// TIA Portal V18 export
FUNCTION_BLOCK "IR_Heater_Control"   // FB17, LAD
TITLE = Description
{ S7_Optimized_Access := 'TRUE' }
VERSION : 0.1
// How to control and set the IR lamp:
// To turn on the IR lamp the machine needs to be started and the doors closed. Heater setpoint should be set from 0-100 "Heater_Setpoint", lamp should be turned on by "Heater_ON_OFF". The lamp will activate only when the certain conditions are meet (position/direction/time).
// 
// Right now, the signal from NOAH is being send when spreading and the permission for the lamp is being keep in the function block for a certain period of time to enable the lamp on the way back.
// 
// E-STOP - always check!
// 
// Modes:
// 0 - Heating Feedbox/Printbox when spreading and executing the heater on the way back from PLC
// 1 - Heating only on the way back from NOAH
// 
// Safety is based only on timer. Hardware protection should be implemented ASAP (contactor controlled by thermal fuse / thermistor to cut off the power if the temperature exceeds certain level).
// 
// Things to implement:
// - Remote temperature sensor(already purchased some time ago).
// - Heater_MathFunction to operate heater better based on the measured results
// - PID control
// 
// Status:
// Filip 14.12.2022: Added modes to give full control to NOAH (Mode 1) or control heater on the way back from PLC (Mode 0)
// stored: AutoNumber true, IsIECCheckEnabled false, IsRetainMemResEnabled false, MemoryReserve 100, SetENOAutomatically false, UDAEnableTagReadback false
   VAR_INPUT
      MachineNumber : Int;
      Mode : Int := 1;   // 0 - Heating partly from PLC; 1 - Full control from NOAH
      DoorSenor : Bool;
      RollerON { ExternalAccessible := 'False'; ExternalVisible := 'False'; ExternalWritable := 'False'} : Bool;   // General heater safety condition
      Heater_Safety_PDL { ExternalAccessible := 'False'; ExternalVisible := 'False'; ExternalWritable := 'False'} : Real;   // Pulse Duration Limit - set by technician or engineer in charge, don't change
      Heater_PWM_address { ExternalAccessible := 'False'; ExternalVisible := 'False'; ExternalWritable := 'False'} : HW_PWM;   // PLC PWM output address
      Heater_Setpoint { ExternalAccessible := 'False'; ExternalVisible := 'False'; ExternalWritable := 'False'} : Real;
      "E-STOP" { ExternalAccessible := 'False'; ExternalVisible := 'False'; ExternalWritable := 'False'} : Bool;
      Heater_ON_OFF { ExternalAccessible := 'False'; ExternalVisible := 'False'; ExternalWritable := 'False'} : Bool;   // WebDB
      FeedboxHeating : Bool;
      PrintboxHeating : Bool;
      AxisYActualPosition : DInt;
      AxisYActualVelocity : Real;
      FeedboxStartMachine : DInt;
      FeedboxEndMachine : DInt;
      PrintboxStartMachine : DInt;
      PrintboxEndMachine : DInt;
      HeaterTest : Bool;
   END_VAR
   VAR_OUTPUT
      Heater_Output : Bool;
      Heater_Pulse_Duration : Int;
      Heater_Error : Int;
      Heater_Output_Check : Int;
      RollerONWayBack : Bool;
      WrongPositionInput : Bool;
   END_VAR
   VAR
      Heater_Scale_LimitReductionBed : Real := 1000.0;   // For big printbox set 70.0, for testing and reduction bed set 100.0
      Heater_Scale_LimitNoReduction : Real := 700.0;
      Heater_Scale_Internal : Real;
      Heater_status : Bool := false;
      Heater_signal : Int;
      Heater_safety_input : Bool := true;   // General heater safety condition
      Heater_error_code : Word;   // Error codes: 0 - OK; 80A1 - Hardware ID; 80D0 - PWM not activated
      Heater_Output_Check_1 : Int;
      SafetyTime : Bool;   // Safety time to not overheat recoater
      ReverseDirectionPermission : Bool := false;   // Permission for using IR on the way back
      ReverseDirection : Bool;
      HeaterStatusSave : Bool;
      HeaterStatusTimeExpired : Bool;
      TurningOnInAdvanceSTART : DInt := 150000;
      TurningOnInAdvanceEND : DInt := 225000;
      TurningOnInAdvanceRefresh : DInt := 2000;
      Position { ExternalAccessible := 'False'; ExternalVisible := 'False'; ExternalWritable := 'False'} : DInt;
      FeedboxHeatingON : Bool := false;
      PrintboxHeatingON : Bool := true;
      HeaterWayBack : Bool := true;
      MaintenanceSkipPositionPermission : Bool;
      MaintenanceSkipRoller : Bool;
      DevModeHeater : Bool;
      DevelopmentAddOn01 : Bool;   // For testing - Will be removed when checked
   END_VAR
   VAR_TEMP
      Heater_SetpointTemp : Int;
      Heater_SetpointOneThird : Int;
      InitialOneThird : Bool;
      Heater_PDLTemp : Int;
      Heater_PDL_conv : Real;
      Heater_Setpoint_Internal01 : Real;
      Heater_Setpoint_Internal02 : Real;
      Heater_Overload : Bool;
      PositionPermissionRight : Bool;
      PositionPermissionLeft : Bool;
      VelocityFactor : Real;
      PositionStartInternal : DInt;
      PositionStartInAdvance : DInt;
      PositionEndInternal : DInt;
      PositionEndInAdvance : DInt;
      PositionEndRefresh : DInt;
      PrintboxSize : DInt;
   END_VAR
   VAR_TEMP   // added for the SCL form of the ladder/FBD networks
      _w1 : Bool;
   END_VAR
BEGIN

REGION Network 1: Safety
   // Heater time safety limitation to avoid overheating parts.
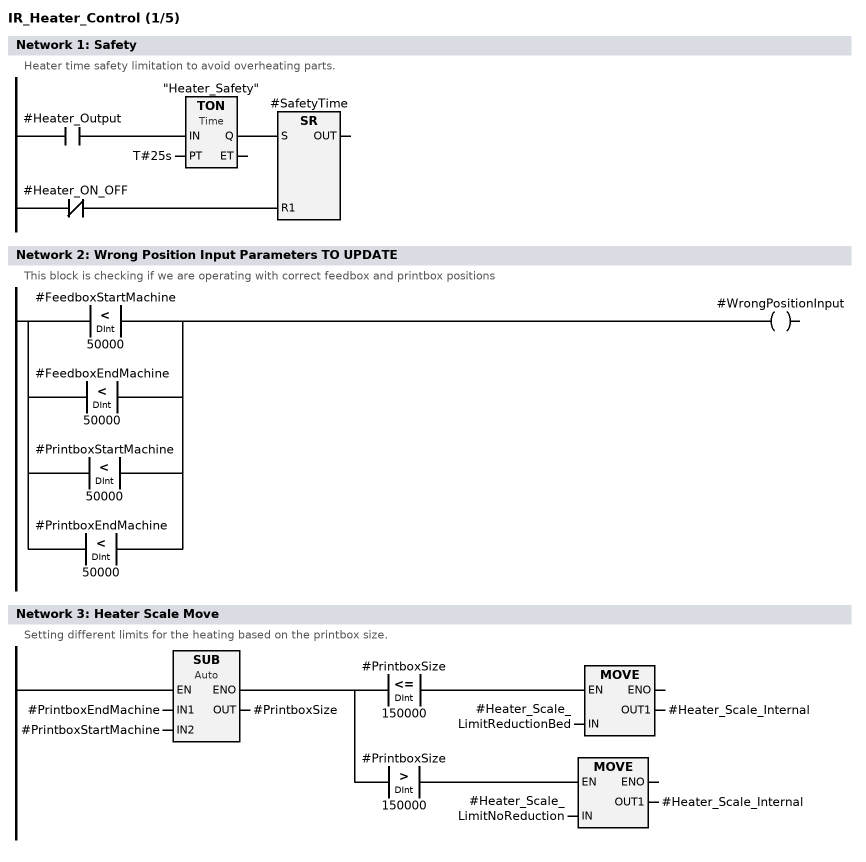
   RUNG wire#powerrail
      Contact( #Heater_Output )
      { S7_Templates := "time_type := Time" } "Heater_Safety".TON(pt := T#25s, et =>)
      S_SR(operand := #SafetyTime, r1 := wire#w1)
   END_RUNG
   RUNG wire#powerrail
      I_Contact( #Heater_ON_OFF )
   END_RUNG wire#w1
   // the same network as SCL:
   "Heater_Safety".TON(IN := #Heater_Output, PT := T#25s);
   IF "Heater_Safety".Q THEN
       #SafetyTime := TRUE;   // SR flip-flop
   END_IF;
   IF NOT #Heater_ON_OFF THEN #SafetyTime := FALSE; END_IF;
END_REGION

REGION Network 2: Wrong Position Input Parameters TO UPDATE
   // This block is checking if we are operating with correct feedbox and printbox positions
   RUNG wire#powerrail
      { S7_Templates := "SrcType := DInt" } LT_Contact(in1 := #FeedboxStartMachine, in2 := 50000)
      wire#w1
      Coil( #WrongPositionInput )
   END_RUNG
   RUNG wire#powerrail
      { S7_Templates := "SrcType := DInt" } LT_Contact(in1 := #FeedboxEndMachine, in2 := 50000)
   END_RUNG wire#w1
   RUNG wire#powerrail
      { S7_Templates := "SrcType := DInt" } LT_Contact(in1 := #PrintboxStartMachine, in2 := 50000)
   END_RUNG wire#w1
   RUNG wire#powerrail
      { S7_Templates := "SrcType := DInt" } LT_Contact(in1 := #PrintboxEndMachine, in2 := 50000)
   END_RUNG wire#w1
   // the same network as SCL:
   #WrongPositionInput := (#FeedboxStartMachine < 50000) OR (#FeedboxEndMachine < 50000) OR (#PrintboxStartMachine < 50000) OR (#PrintboxEndMachine < 50000);
END_REGION

REGION Network 3: Heater Scale Move
   // Setting different limits for the heating based on the printbox size.
   RUNG wire#powerrail
      Sub(in1 := #PrintboxEndMachine, in2 := #PrintboxStartMachine, out => #PrintboxSize)
      wire#w1
      { S7_Templates := "SrcType := DInt" } LE_Contact(in1 := #PrintboxSize, in2 := 150000)
      Move(in := #Heater_Scale_LimitReductionBed, out1 => #Heater_Scale_Internal)
   END_RUNG
   RUNG wire#w1
      { S7_Templates := "SrcType := DInt" } GT_Contact(in1 := #PrintboxSize, in2 := 150000)
      Move(in := #Heater_Scale_LimitNoReduction, out1 => #Heater_Scale_Internal)
   END_RUNG
   // the same network as SCL:
   #PrintboxSize := #PrintboxEndMachine - #PrintboxStartMachine;
   IF #PrintboxSize <= 150000 THEN #Heater_Scale_Internal := #Heater_Scale_LimitReductionBed; END_IF;
   IF #PrintboxSize > 150000 THEN #Heater_Scale_Internal := #Heater_Scale_LimitNoReduction; END_IF;
END_REGION

REGION Network 4: Positions In Advance
   // Calculation of positions to turn on IR lamp in advance, due to long rise time.
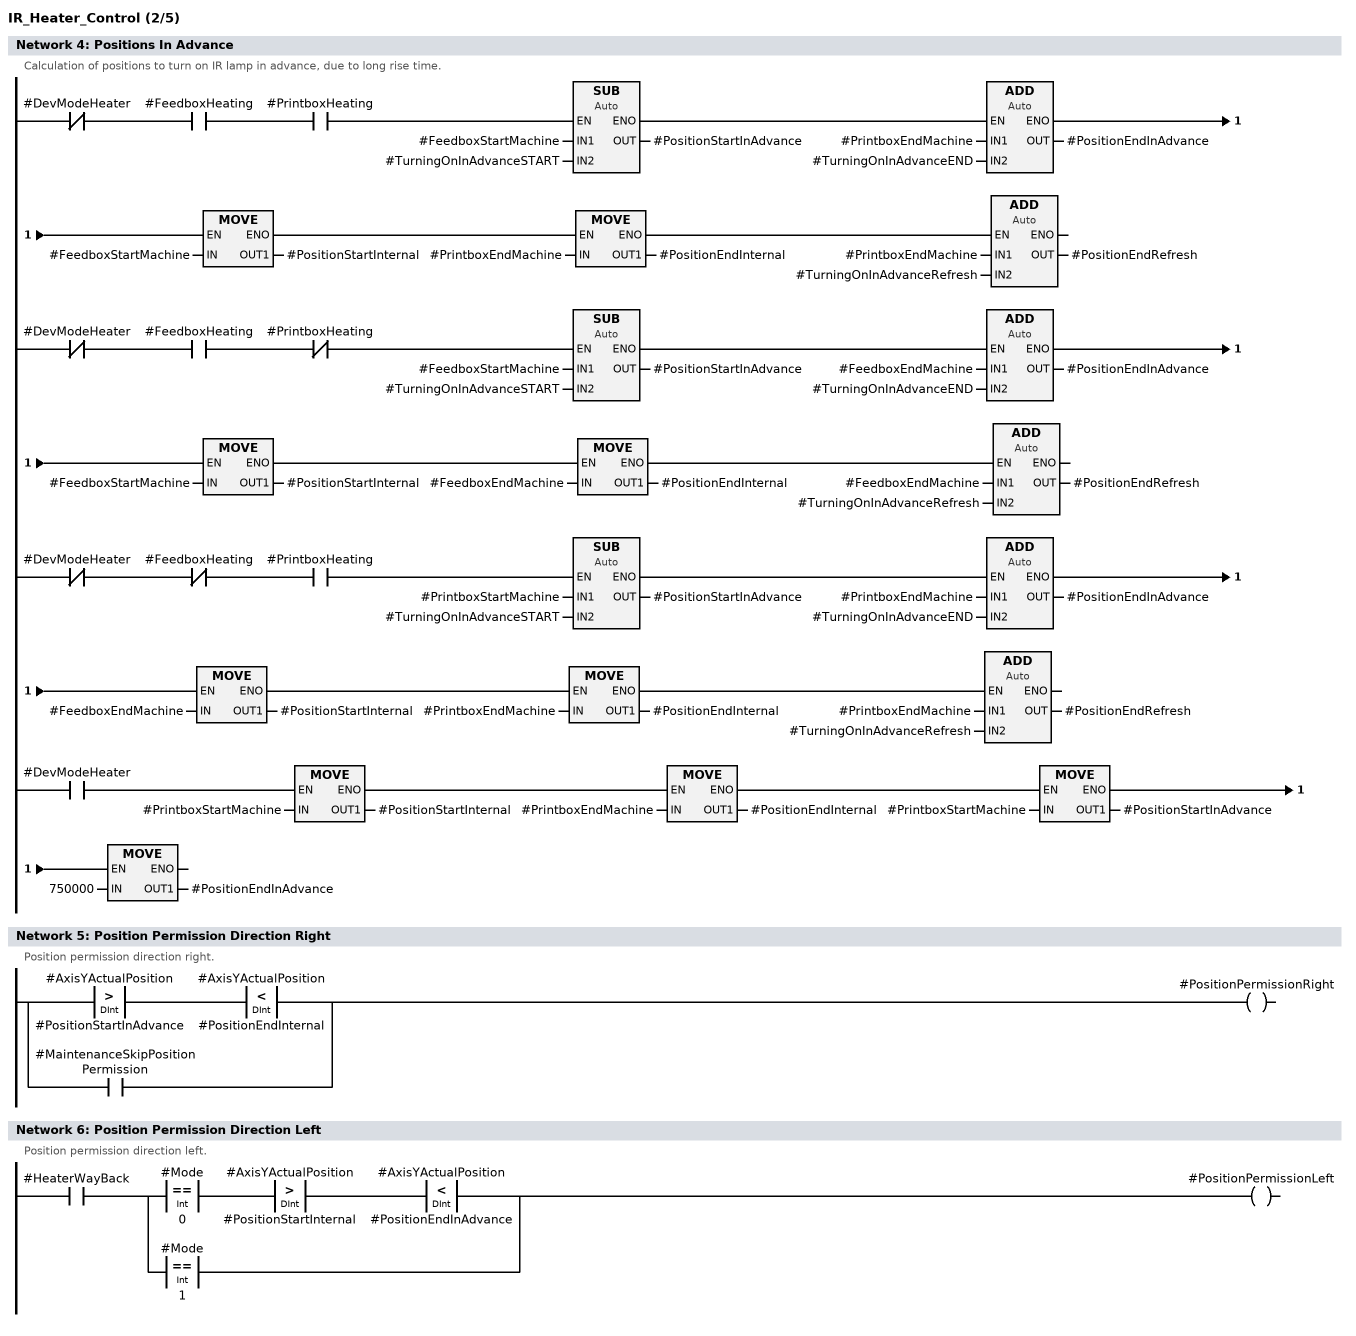
   RUNG wire#powerrail
      I_Contact( #DevModeHeater )
      Contact( #FeedboxHeating )
      Contact( #PrintboxHeating )
      Sub(in1 := #FeedboxStartMachine, in2 := #TurningOnInAdvanceSTART, out => #PositionStartInAdvance)
      Add(in1 := #PrintboxEndMachine, in2 := #TurningOnInAdvanceEND, out => #PositionEndInAdvance)
      Move(in := #FeedboxStartMachine, out1 => #PositionStartInternal)
      Move(in := #PrintboxEndMachine, out1 => #PositionEndInternal)
      Add(in1 := #PrintboxEndMachine, in2 := #TurningOnInAdvanceRefresh, out => #PositionEndRefresh)
   END_RUNG
   RUNG wire#powerrail
      I_Contact( #DevModeHeater )
      Contact( #FeedboxHeating )
      I_Contact( #PrintboxHeating )
      Sub(in1 := #FeedboxStartMachine, in2 := #TurningOnInAdvanceSTART, out => #PositionStartInAdvance)
      Add(in1 := #FeedboxEndMachine, in2 := #TurningOnInAdvanceEND, out => #PositionEndInAdvance)
      Move(in := #FeedboxStartMachine, out1 => #PositionStartInternal)
      Move(in := #FeedboxEndMachine, out1 => #PositionEndInternal)
      Add(in1 := #FeedboxEndMachine, in2 := #TurningOnInAdvanceRefresh, out => #PositionEndRefresh)
   END_RUNG
   RUNG wire#powerrail
      I_Contact( #DevModeHeater )
      I_Contact( #FeedboxHeating )
      Contact( #PrintboxHeating )
      Sub(in1 := #PrintboxStartMachine, in2 := #TurningOnInAdvanceSTART, out => #PositionStartInAdvance)
      Add(in1 := #PrintboxEndMachine, in2 := #TurningOnInAdvanceEND, out => #PositionEndInAdvance)
      Move(in := #FeedboxEndMachine, out1 => #PositionStartInternal)
      Move(in := #PrintboxEndMachine, out1 => #PositionEndInternal)
      Add(in1 := #PrintboxEndMachine, in2 := #TurningOnInAdvanceRefresh, out => #PositionEndRefresh)
   END_RUNG
   RUNG wire#powerrail
      Contact( #DevModeHeater )
      Move(in := #PrintboxStartMachine, out1 => #PositionStartInternal)
      Move(in := #PrintboxEndMachine, out1 => #PositionEndInternal)
      Move(in := #PrintboxStartMachine, out1 => #PositionStartInAdvance)
      Move(in := 750000, out1 => #PositionEndInAdvance)
   END_RUNG
   // the same network as SCL:
   IF NOT #DevModeHeater AND #FeedboxHeating AND #PrintboxHeating THEN
       #PositionStartInAdvance := #FeedboxStartMachine - #TurningOnInAdvanceSTART;
       #PositionEndInAdvance := #PrintboxEndMachine + #TurningOnInAdvanceEND;
       #PositionStartInternal := #FeedboxStartMachine;
       #PositionEndInternal := #PrintboxEndMachine;
       #PositionEndRefresh := #PrintboxEndMachine + #TurningOnInAdvanceRefresh;
   END_IF;
   IF NOT #DevModeHeater AND #FeedboxHeating AND NOT #PrintboxHeating THEN
       #PositionStartInAdvance := #FeedboxStartMachine - #TurningOnInAdvanceSTART;
       #PositionEndInAdvance := #FeedboxEndMachine + #TurningOnInAdvanceEND;
       #PositionStartInternal := #FeedboxStartMachine;
       #PositionEndInternal := #FeedboxEndMachine;
       #PositionEndRefresh := #FeedboxEndMachine + #TurningOnInAdvanceRefresh;
   END_IF;
   IF NOT #DevModeHeater AND NOT #FeedboxHeating AND #PrintboxHeating THEN
       #PositionStartInAdvance := #PrintboxStartMachine - #TurningOnInAdvanceSTART;
       #PositionEndInAdvance := #PrintboxEndMachine + #TurningOnInAdvanceEND;
       #PositionStartInternal := #FeedboxEndMachine;
       #PositionEndInternal := #PrintboxEndMachine;
       #PositionEndRefresh := #PrintboxEndMachine + #TurningOnInAdvanceRefresh;
   END_IF;
   IF #DevModeHeater THEN
       #PositionStartInternal := #PrintboxStartMachine;
       #PositionEndInternal := #PrintboxEndMachine;
       #PositionStartInAdvance := #PrintboxStartMachine;
       #PositionEndInAdvance := 750000;
   END_IF;
END_REGION

REGION Network 5: Position Permission Direction Right
   // Position permission direction right.
   RUNG wire#powerrail
      { S7_Templates := "SrcType := DInt" } GT_Contact(in1 := #AxisYActualPosition, in2 := #PositionStartInAdvance)
      { S7_Templates := "SrcType := DInt" } LT_Contact(in1 := #AxisYActualPosition, in2 := #PositionEndInternal)
      wire#w1
      Coil( #PositionPermissionRight )
   END_RUNG
   RUNG wire#powerrail
      Contact( #MaintenanceSkipPositionPermission )
   END_RUNG wire#w1
   // the same network as SCL:
   #PositionPermissionRight := ((#AxisYActualPosition > #PositionStartInAdvance) AND (#AxisYActualPosition < #PositionEndInternal)) OR #MaintenanceSkipPositionPermission;
END_REGION

REGION Network 6: Position Permission Direction Left
   // Position permission direction left.
   RUNG wire#powerrail
      Contact( #HeaterWayBack )
      wire#w1
      { S7_Templates := "SrcType := Int" } EQ_Contact(in1 := #Mode, in2 := 0)
      { S7_Templates := "SrcType := DInt" } GT_Contact(in1 := #AxisYActualPosition, in2 := #PositionStartInternal)
      { S7_Templates := "SrcType := DInt" } LT_Contact(in1 := #AxisYActualPosition, in2 := #PositionEndInAdvance)
      wire#w2
      Coil( #PositionPermissionLeft )
   END_RUNG
   RUNG wire#w1
      { S7_Templates := "SrcType := Int" } EQ_Contact(in1 := #Mode, in2 := 1)
   END_RUNG wire#w2
   // the same network as SCL:
   #PositionPermissionLeft := #HeaterWayBack AND (((#Mode = 0) AND (#AxisYActualPosition > #PositionStartInternal) AND (#AxisYActualPosition < #PositionEndInAdvance)) OR (#Mode = 1));
END_REGION

REGION Network 7: Reverse Direction for Armadillo V6
   // Detection of the reverse direction of the Y axis motion.
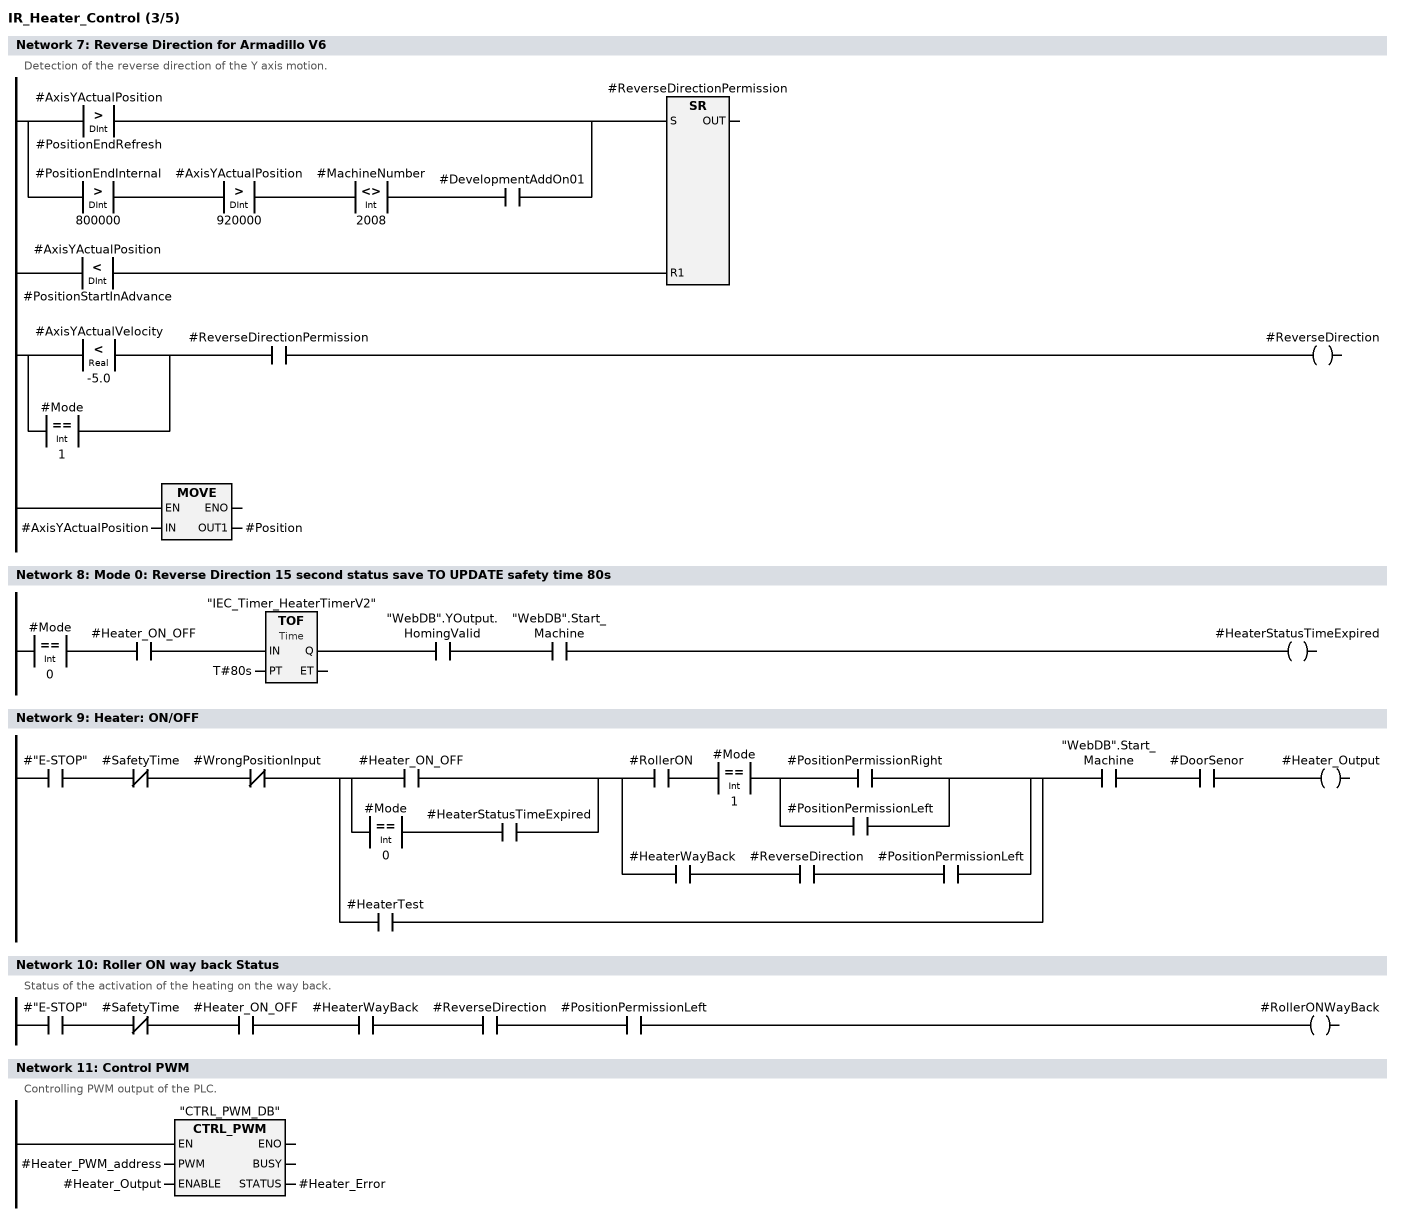
   RUNG wire#powerrail
      { S7_Templates := "SrcType := DInt" } GT_Contact(in1 := #AxisYActualPosition, in2 := #PositionEndRefresh)
      wire#w1
      S_SR(operand := #ReverseDirectionPermission, r1 := wire#w2)
   END_RUNG
   RUNG wire#powerrail
      { S7_Templates := "SrcType := DInt" } GT_Contact(in1 := #PositionEndInternal, in2 := 800000)
      { S7_Templates := "SrcType := DInt" } GT_Contact(in1 := #AxisYActualPosition, in2 := 920000)
      { S7_Templates := "SrcType := Int" } NE_Contact(in1 := #MachineNumber, in2 := 2008)
      Contact( #DevelopmentAddOn01 )
   END_RUNG wire#w1
   RUNG wire#powerrail
      { S7_Templates := "SrcType := DInt" } LT_Contact(in1 := #AxisYActualPosition, in2 := #PositionStartInAdvance)
   END_RUNG wire#w2
   RUNG wire#powerrail
      { S7_Templates := "SrcType := Real" } LT_Contact(in1 := #AxisYActualVelocity, in2 := -5.0)
      wire#w3
      Contact( #ReverseDirectionPermission )
      Coil( #ReverseDirection )
   END_RUNG
   RUNG wire#powerrail
      { S7_Templates := "SrcType := Int" } EQ_Contact(in1 := #Mode, in2 := 1)
   END_RUNG wire#w3
   RUNG wire#powerrail
      Move(in := #AxisYActualPosition, out1 => #Position)
   END_RUNG
   // the same network as SCL:
   IF (#AxisYActualPosition > #PositionEndRefresh) OR ((#PositionEndInternal > 800000) AND (#AxisYActualPosition > 920000) AND (#MachineNumber <> 2008) AND #DevelopmentAddOn01) THEN
       #ReverseDirectionPermission := TRUE;   // SR flip-flop
   END_IF;
   IF #AxisYActualPosition < #PositionStartInAdvance THEN #ReverseDirectionPermission := FALSE; END_IF;
   #ReverseDirection := ((#AxisYActualVelocity < (-5.0)) OR (#Mode = 1)) AND #ReverseDirectionPermission;
   #Position := #AxisYActualPosition;
END_REGION

REGION Network 8: Mode 0: Reverse Direction 15 second status save TO UPDATE safety time 80s
   RUNG wire#powerrail
      { S7_Templates := "SrcType := Int" } EQ_Contact(in1 := #Mode, in2 := 0)
      Contact( #Heater_ON_OFF )
      { S7_Templates := "time_type := Time" } "IEC_Timer_HeaterTimerV2".TOF(pt := T#80s, et =>)
      Contact( "WebDB".YOutput.HomingValid )
      Contact( "WebDB".Start_Machine )
      Coil( #HeaterStatusTimeExpired )
   END_RUNG
   // the same network as SCL:
   "IEC_Timer_HeaterTimerV2".TOF(IN := (#Mode = 0) AND #Heater_ON_OFF, PT := T#80s);
   #HeaterStatusTimeExpired := "IEC_Timer_HeaterTimerV2".Q AND "WebDB".YOutput.HomingValid AND "WebDB".Start_Machine;
END_REGION

REGION Network 9: Heater: ON/OFF
   RUNG wire#powerrail
      Contact( #"E-STOP" )
      I_Contact( #SafetyTime )
      I_Contact( #WrongPositionInput )
      wire#w1
      Contact( #Heater_ON_OFF )
      wire#w2
      Contact( #RollerON )
      { S7_Templates := "SrcType := Int" } EQ_Contact(in1 := #Mode, in2 := 1)
      wire#w3
      Contact( #PositionPermissionRight )
      wire#w4
      Contact( "WebDB".Start_Machine )
      Contact( #DoorSenor )
      Coil( #Heater_Output )
   END_RUNG
   RUNG wire#w1
      { S7_Templates := "SrcType := Int" } EQ_Contact(in1 := #Mode, in2 := 0)
      Contact( #HeaterStatusTimeExpired )
   END_RUNG wire#w2
   RUNG wire#w3
      Contact( #PositionPermissionLeft )
   END_RUNG wire#w4
   RUNG wire#w2
      Contact( #HeaterWayBack )
      Contact( #ReverseDirection )
      Contact( #PositionPermissionLeft )
   END_RUNG wire#w4
   RUNG wire#w1
      Contact( #HeaterTest )
   END_RUNG wire#w4
   // the same network as SCL:
   #Heater_Output := #"E-STOP" AND NOT #SafetyTime AND NOT #WrongPositionInput AND (((#Heater_ON_OFF OR ((#Mode = 0) AND #HeaterStatusTimeExpired)) AND ((#RollerON AND (#Mode = 1) AND (#PositionPermissionRight OR #PositionPermissionLeft)) OR (#HeaterWayBack AND #ReverseDirection AND #PositionPermissionLeft))) OR #HeaterTest) AND "WebDB".Start_Machine AND #DoorSenor;
END_REGION

REGION Network 10: Roller ON way back Status
   // Status of the activation of the heating on the way back.
   RUNG wire#powerrail
      Contact( #"E-STOP" )
      I_Contact( #SafetyTime )
      Contact( #Heater_ON_OFF )
      Contact( #HeaterWayBack )
      Contact( #ReverseDirection )
      Contact( #PositionPermissionLeft )
      Coil( #RollerONWayBack )
   END_RUNG
   // the same network as SCL:
   #RollerONWayBack := #"E-STOP" AND NOT #SafetyTime AND #Heater_ON_OFF AND #HeaterWayBack AND #ReverseDirection AND #PositionPermissionLeft;
END_REGION

REGION Network 11: Control PWM
   // Controlling PWM output of the PLC.
   RUNG wire#powerrail
      "CTRL_PWM_DB".CTRL_PWM(PWM := #Heater_PWM_address, ENABLE := #Heater_Output, BUSY =>, STATUS => #Heater_Error)
   END_RUNG
   // the same network as SCL:
   "CTRL_PWM_DB"(PWM := #Heater_PWM_address, ENABLE := #Heater_Output, STATUS => #Heater_Error);   // CTRL_PWM
END_REGION

REGION Network 12: Conversion
   // Conversion of the heater setpoint and limit.
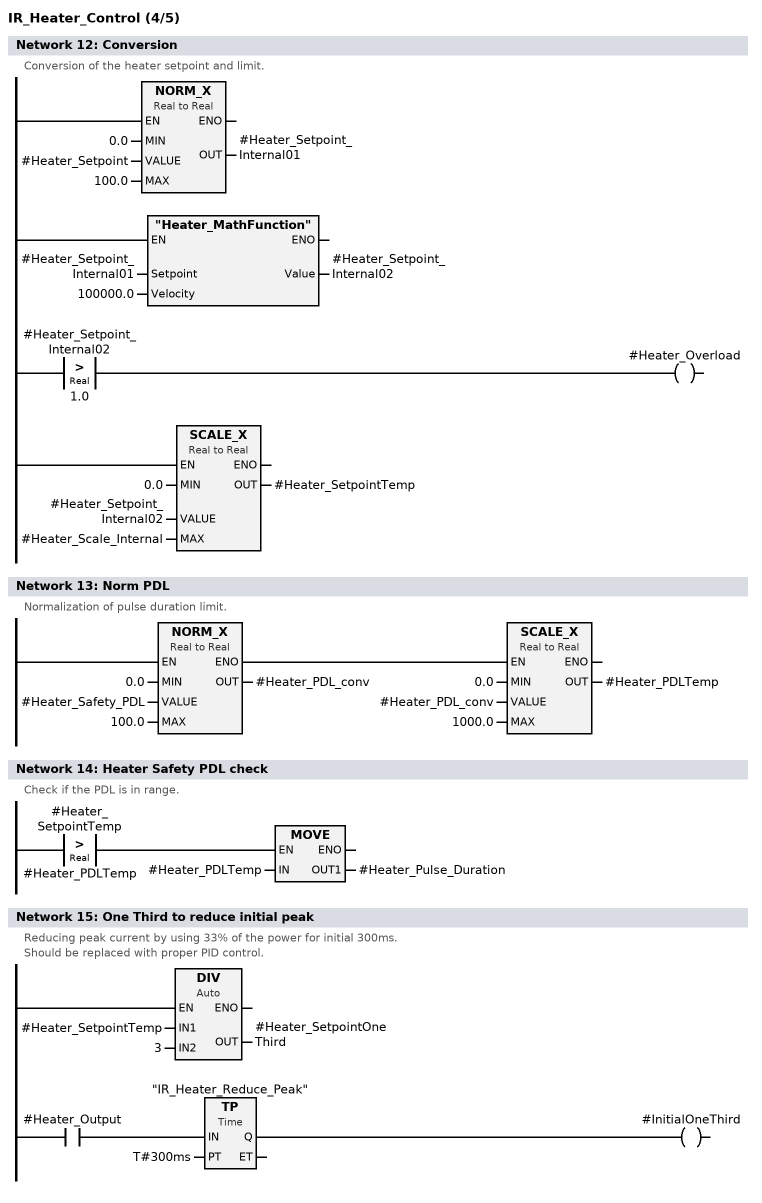
   RUNG wire#powerrail
      { S7_Templates := "[SrcType := Real, DestType := Real]" } Normalize(min := 0.0, value := #Heater_Setpoint, max := 100.0, out => #Heater_Setpoint_Internal01)
   END_RUNG
   RUNG wire#powerrail
      "Heater_MathFunction"(Setpoint := #Heater_Setpoint_Internal01, Velocity := 100000.0, Value => #Heater_Setpoint_Internal02)
   END_RUNG
   RUNG wire#powerrail
      { S7_Templates := "SrcType := Real" } GT_Contact(in1 := #Heater_Setpoint_Internal02, in2 := 1.0)
      Coil( #Heater_Overload )
   END_RUNG
   RUNG wire#powerrail
      { S7_Templates := "[SrcType := Real, DestType := Real]" } Scale(min := 0.0, value := #Heater_Setpoint_Internal02, max := #Heater_Scale_Internal, out => #Heater_SetpointTemp)
   END_RUNG
   // the same network as SCL:
   #Heater_Setpoint_Internal01 := NORM_X(MIN := 0.0, VALUE := #Heater_Setpoint, MAX := 100.0);
   "Heater_MathFunction"(Setpoint := #Heater_Setpoint_Internal01,
                         Velocity := 100000.0,
                         Value => #Heater_Setpoint_Internal02);
   #Heater_Overload := #Heater_Setpoint_Internal02 > 1.0;
   #Heater_SetpointTemp := SCALE_X(MIN := 0.0, VALUE := #Heater_Setpoint_Internal02, MAX := #Heater_Scale_Internal);
END_REGION

REGION Network 13: Norm PDL
   // Normalization of pulse duration limit.
   RUNG wire#powerrail
      { S7_Templates := "[SrcType := Real, DestType := Real]" } Normalize(min := 0.0, value := #Heater_Safety_PDL, max := 100.0, out => #Heater_PDL_conv)
      { S7_Templates := "[SrcType := Real, DestType := Real]" } Scale(min := 0.0, value := #Heater_PDL_conv, max := 1000.0, out => #Heater_PDLTemp)
   END_RUNG
   // the same network as SCL:
   #Heater_PDL_conv := NORM_X(MIN := 0.0, VALUE := #Heater_Safety_PDL, MAX := 100.0);
   #Heater_PDLTemp := SCALE_X(MIN := 0.0, VALUE := #Heater_PDL_conv, MAX := 1000.0);
END_REGION

REGION Network 14: Heater Safety PDL check
   // Check if the PDL is in range.
   RUNG wire#powerrail
      { S7_Templates := "SrcType := Real" } GT_Contact(in1 := #Heater_SetpointTemp, in2 := #Heater_PDLTemp)
      Move(in := #Heater_PDLTemp, out1 => #Heater_Pulse_Duration)
   END_RUNG
   // the same network as SCL:
   IF #Heater_SetpointTemp > #Heater_PDLTemp THEN #Heater_Pulse_Duration := #Heater_PDLTemp; END_IF;
END_REGION

REGION Network 15: One Third to reduce initial peak
   // Reducing peak current by using 33% of the power for initial 300ms.
   // 
   // Should be replaced with proper PID control.
   RUNG wire#powerrail
      Div(in1 := #Heater_SetpointTemp, in2 := 3, out => #Heater_SetpointOneThird)
   END_RUNG
   RUNG wire#powerrail
      Contact( #Heater_Output )
      { S7_Templates := "time_type := Time" } "IR_Heater_Reduce_Peak".TP(pt := T#300ms, et =>)
      Coil( #InitialOneThird )
   END_RUNG
   // the same network as SCL:
   #Heater_SetpointOneThird := #Heater_SetpointTemp / 3;
   "IR_Heater_Reduce_Peak".TP(IN := #Heater_Output, PT := T#300ms);
   #InitialOneThird := "IR_Heater_Reduce_Peak".Q;
END_REGION

REGION Network 16: Move
   // Moving heating parameters.
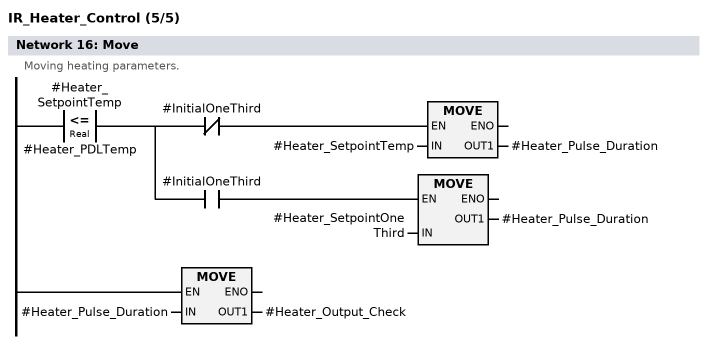
   RUNG wire#powerrail
      { S7_Templates := "SrcType := Real" } LE_Contact(in1 := #Heater_SetpointTemp, in2 := #Heater_PDLTemp)
      wire#w1
      I_Contact( #InitialOneThird )
      Move(in := #Heater_SetpointTemp, out1 => #Heater_Pulse_Duration)
   END_RUNG
   RUNG wire#w1
      Contact( #InitialOneThird )
      Move(in := #Heater_SetpointOneThird, out1 => #Heater_Pulse_Duration)
   END_RUNG
   RUNG wire#powerrail
      Move(in := #Heater_Pulse_Duration, out1 => #Heater_Output_Check)
   END_RUNG
   // the same network as SCL:
   #_w1 := #Heater_SetpointTemp <= #Heater_PDLTemp;
   IF #_w1 AND NOT #InitialOneThird THEN #Heater_Pulse_Duration := #Heater_SetpointTemp; END_IF;
   IF #_w1 AND #InitialOneThird THEN #Heater_Pulse_Duration := #Heater_SetpointOneThird; END_IF;
   #Heater_Output_Check := #Heater_Pulse_Duration;
END_REGION
END_FUNCTION_BLOCK
